FUNCTION_BLOCK FutureGripperControlCreator IMPLEMENTS InterfaceTaskCreator
VAR_INPUT
END_VAR
VAR_OUTPUT
END_VAR
VAR
	_gripper_close_output : REFERENCE TO BOOL;
	_gripper_open_output : REFERENCE TO BOOL;
	_gripper_closed_sensor : REFERENCE TO BOOL;
	_gripper_open_sensor : REFERENCE TO BOOL;
	_command : BOOL;
	_timeout : TIME := T#5S;
END_VAR

METHOD create_future : InterfaceFuture
VAR_INPUT
    future_name : STRING;
END_VAR
VAR
    _p_future : POINTER TO FutureGripperControl;
END_VAR
_p_future := __NEW(FutureGripperControl);
_p_future^.future_name := future_name;

_p_future^.set_parameters(
    gripper_close_output := _gripper_close_output,
    gripper_open_output := _gripper_open_output,
    gripper_closed_sensor := _gripper_closed_sensor,
    gripper_open_sensor := _gripper_open_sensor,
    command := _command,
    timeout := _timeout
);

create_future := _p_future^;
END_METHOD

METHOD destroy_future : InterfaceFuture
VAR_INPUT
    future : InterfaceFuture;
END_VAR
VAR
    _p_future : POINTER TO FutureGripperControl;
END_VAR
IF __QUERYPOINTER(future, _p_future) THEN
	__DELETE(_p_future);
	IF _p_future = 0 THEN
		destroy_future := 0;
	END_IF
END_IF
END_METHOD

METHOD set_parameters : BOOL
VAR_INPUT
	gripper_close_output : REFERENCE TO BOOL;
	gripper_open_output : REFERENCE TO BOOL;
	gripper_closed_sensor : REFERENCE TO BOOL;
	gripper_open_sensor : REFERENCE TO BOOL;
	command : BOOL;
	timeout : TIME := T#5S;
END_VAR
_gripper_close_output REF= gripper_close_output;
_gripper_open_output REF= gripper_open_output;
_gripper_closed_sensor REF= gripper_closed_sensor;
_gripper_open_sensor REF= gripper_open_sensor;
_command := command;
_timeout := timeout;
set_parameters := TRUE;
END_METHOD

END_FUNCTION_BLOCK

(* stored: Version 1.1.0.1, ProductVersion 3.1.4024.12
   POU FutureGripperControlCreator: Id {87654321-4321-4321-4321-123456789abc}, SpecialFunc None
   Method create_future: Id {87654321-4321-4321-4321-123456789def}
   Method destroy_future: Id {87654321-4321-4321-4321-123456789fed}
   Method set_parameters: Id {87654321-4321-4321-4321-123456789cba} *)
